Fanuc KAREL source: kt00982.KL

PROGRAM KT00982
%STACKSIZE=65535
%PRIORITY=65535
%NOLOCKGROUP
VAR
R1 : REAL
R2 : REAL
OUT : POSITION
-- UNRESOLVED DECLARATIONS (source type spelling not recovered)
-- CFG : TYPE_0x001C (type_u16=0x001C)
BEGIN
R1=2.0
R2=3.0
R1=2.0
R2=3.0
-- UNRESOLVED_PC line 13 opcodes [9D 22 A5] marker_code=64
-- UNRESOLVED_PC line 14 opcodes [27 22 22 22 22 22 22 22 76 7E 4A] marker_code=79
END KT00982
